FUNCTION_BLOCK FB_Display IMPLEMENTS ITF_Observer
VAR
	data : INT; //updated from the Observable
	_ID	 : udint; //set by the Observable
END_VAR

METHOD CyclicLogic : BOOL
VAR_INPUT
END_VAR
END_METHOD

PROPERTY ID : udint
GET
ID := _ID;
END_GET
SET
_ID := ID;
END_SET
END_PROPERTY

METHOD update : BOOL
VAR_INPUT
	Station : REFERENCE TO FB_Station;
END_VAR
data := Station.Data; //Read what you want from the Observable4
END_METHOD

END_FUNCTION_BLOCK

(* stored: Version 1.1.0.1, ProductVersion 3.1.4024.12
   POU FB_Display: Id {c38be1ce-6876-4ccb-9de3-5bab7019eeb4}, SpecialFunc None
   Folder ITF_Observer: Id {fcd202ed-2f65-495c-8a88-96ce17698f1a}
   Method CyclicLogic: Id {8448c9a2-d7c2-48a0-8215-62dd23a0a229}
   Property ID: Id {ab153b6e-3229-4478-97b7-d3ef9a95b506}
   Get Get: Id {efb636fa-abc1-48b8-93ba-bfa504f73b3e}
   Set Set: Id {62312570-e819-4d42-9bc5-fbf0a42d00fc}
   Method update: Id {9c98bc60-509f-478e-89e7-5a747d53d700} *)
